FUNCTION_BLOCK TcoCylinderMoveTask EXTENDS TcoCore.TcoTask
VAR_INPUT
	PositionSensor		   : BOOL;
	MaxTimeToReachPosition : TIME := T#10S;
	TimeToRefill 		   : TIME := T#100MS;
	PositionName		   : STRING(25);
	refInverseTask: REFERENCE TO TcoCore.TcoTask;
END_VAR
VAR_IN_OUT
	MoveToPositionSignal : BOOL;
	InverseSignal		 : BOOL;	
END_VAR

VAR
	_stringBuilder : TcoCore.StringBuilder;
END_VAR

IF (THIS^.Execute()) THEN
	IF(THIS^.ElapsedTime > MaxTimeToReachPosition) THEN THIS^.Messenger.Warning(_stringBuilder.Clear().Append(PositionName).Append(' sensor not reached yet.').ToString()); END_IF;
	InverseSignal		 := FALSE;
	MoveToPositionSignal := TRUE;
	THIS^.DoneWhen(PositionSensor);	
END_IF

METHOD PUBLIC FB_init : BOOL
VAR_INPUT
	bInitRetains : BOOL; // if TRUE, the retain variables are initialized (warm start / cold start)
	bInCopyCode : BOOL;  // if TRUE, the instance afterwards gets moved into the copy code (online change)
	ParentObject : ITcoObject;	
END_VAR
END_METHOD

(*~
	<docu>
		<summary>
			Executes when task is aborted.
		</summary>			
	</docu>	
~*)
METHOD PROTECTED OnAbort
MoveToPositionSignal := FALSE;
END_METHOD

METHOD PROTECTED OnError
END_METHOD

METHOD PROTECTED OnStart
IF __ISVALIDREF(refInverseTask) THEN
	refInverseTask.Restore();
END_IF
END_METHOD

END_FUNCTION_BLOCK

(* stored: Version 1.1.0.1, ProductVersion 3.1.4024.12
   POU TcoCylinderMoveTask: Id {36f82742-ef83-064d-3f82-8df2b1eb7a0b}, SpecialFunc None
   Method FB_init: Id {cf5faab0-ae9a-0dcc-0a9f-d4a07856e2e1}
   Method OnAbort: Id {45e7f28e-39ff-01a9-2b80-1e7ac1ea429e}
   Method OnError: Id {c702604b-83ae-0ede-324b-55447818c6ba}
   Method OnStart: Id {e7f01650-89d3-0bc5-17a1-230c301d4988} *)
